REGION Network 68: **** 4.6 - Machine status - Indications **** Max Bodies HMI - Static
   #H_BodyCounterDynamic.H_StaticMax[1].H_DInt := #I_MaxBody;
END_REGION

REGION Network 69: **** 4.6 - Machine status - Indications **** Dynamic Max Bodies HMI - Dynamic
   #H_BodyCounterDynamic.H_DynamicMax[1].H_DInt := #MaxDynamicBody;
END_REGION

REGION Network 70: **** 4.6 - Machine Status - Indication **** Icon Animation
   IF "TRUE" THEN
       "LSimpleIAnim"(I_SetPos := "TRUE",
                      I_ResetPos := "FALSE",
                      I_Active := "FALSE",
                      I_Invisible := "FALSE",
                      I_OutOfUse := "FALSE",
                      I_AlarmA := "FALSE",
                      I_AlarmB := "FALSE",
                      I_AlarmC := #CounterConv1Fault OR #CounterConv2Fault,
                      I_AlarmD := "FALSE",
                      I_ManualMode := "FALSE",
                      I_FncSelInHMI := "FALSE",
                      H_IAnim => #H_HMI.H_IAnim);
   END_IF;
END_REGION

REGION Network 71: **** 4.6 - Machine status - Indications **** Animation
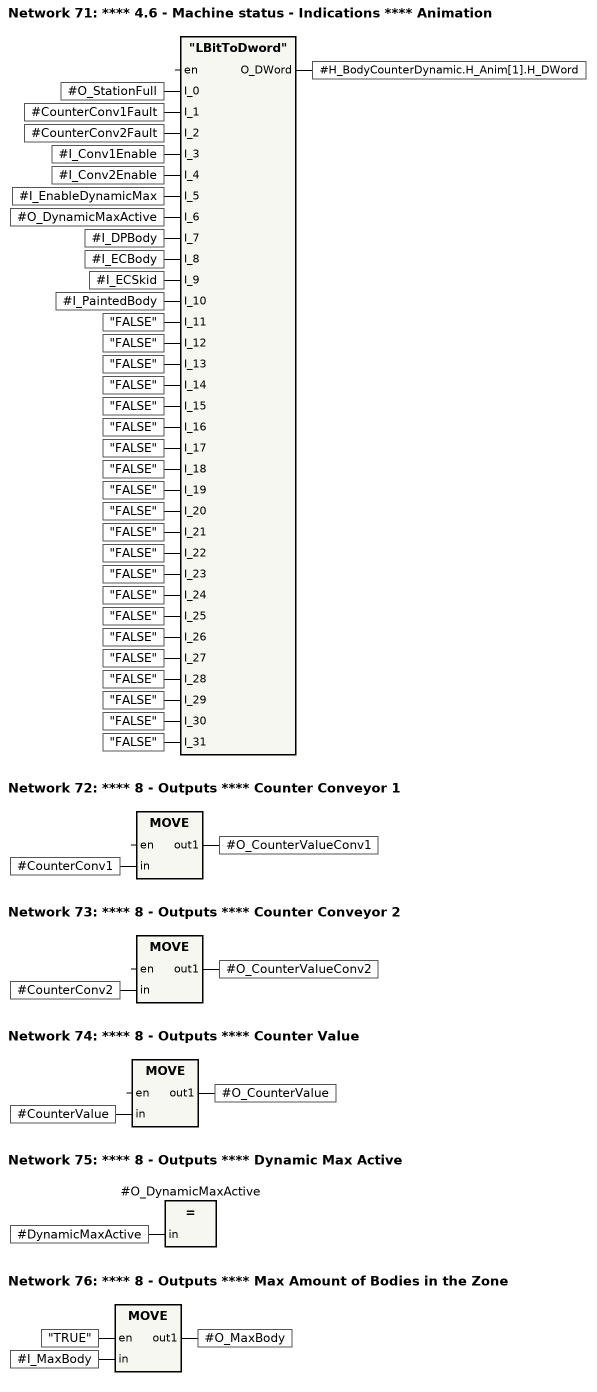
   "LBitToDword"(I_0 := #O_StationFull,
                 I_1 := #CounterConv1Fault,
                 I_2 := #CounterConv2Fault,
                 I_3 := #I_Conv1Enable,
                 I_4 := #I_Conv2Enable,
                 I_5 := #I_EnableDynamicMax,
                 I_6 := #O_DynamicMaxActive,
                 I_7 := #I_DPBody,
                 I_8 := #I_ECBody,
                 I_9 := #I_ECSkid,
                 I_10 := #I_PaintedBody,
                 I_11 := "FALSE",
                 I_12 := "FALSE",
                 I_13 := "FALSE",
                 I_14 := "FALSE",
                 I_15 := "FALSE",
                 I_16 := "FALSE",
                 I_17 := "FALSE",
                 I_18 := "FALSE",
                 I_19 := "FALSE",
                 I_20 := "FALSE",
                 I_21 := "FALSE",
                 I_22 := "FALSE",
                 I_23 := "FALSE",
                 I_24 := "FALSE",
                 I_25 := "FALSE",
                 I_26 := "FALSE",
                 I_27 := "FALSE",
                 I_28 := "FALSE",
                 I_29 := "FALSE",
                 I_30 := "FALSE",
                 I_31 := "FALSE",
                 O_DWord => #H_BodyCounterDynamic.H_Anim[1].H_DWord);
END_REGION

REGION Network 72: **** 8 - Outputs **** Counter Conveyor 1
   #O_CounterValueConv1 := #CounterConv1;
END_REGION

REGION Network 73: **** 8 - Outputs **** Counter Conveyor 2
   #O_CounterValueConv2 := #CounterConv2;
END_REGION

REGION Network 74: **** 8 - Outputs **** Counter Value
   #O_CounterValue := #CounterValue;
END_REGION

REGION Network 75: **** 8 - Outputs **** Dynamic Max Active
   #O_DynamicMaxActive := #DynamicMaxActive;
END_REGION

REGION Network 76: **** 8 - Outputs **** Max Amount of Bodies in the Zone
   IF "TRUE" THEN #O_MaxBody := #I_MaxBody; END_IF;
END_REGION

REGION Network 77: **** 9.1 - Alarm Output **** Counter Conveyor 1 Alarm
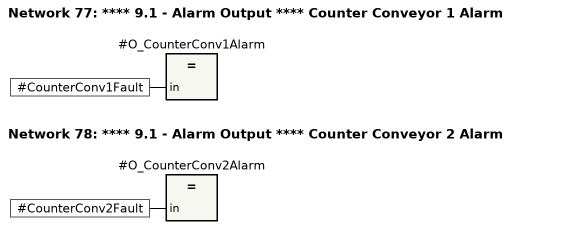
   #O_CounterConv1Alarm := #CounterConv1Fault;
END_REGION

REGION Network 78: **** 9.1 - Alarm Output **** Counter Conveyor 2 Alarm
   #O_CounterConv2Alarm := #CounterConv2Fault;
END_REGION
END_FUNCTION_BLOCK
